{attribute addProperty BoxType "EK1122-0000-0018"}
{attribute addProperty Id "Beckhoff_EL30xxsub_EK1100EK1100_179A0949162"}
{attribute addProperty CRC "3537379036"}
{attribute addProperty SizeInBites "16"}
{attribute addProperty SizeInBytes "2"}
TYPE Beckhoff_EL30xxEK1122_D2D81EDC EXTENDS EK1122_179A0949 :
STRUCT
	{attribute addProperty Name "Beckhoff_EL30xxsub_EK1100"}
	Beckhoff_EL30xxsub_EK1100 : EK1100_179A0949;
END_STRUCT
END_TYPE

(* stored: Version 1.2.0.0, ProductVersion 3.1.4024.9
   DUT Beckhoff_EL30xxEK1122_D2D81EDC: Id {61a4f517-b592-48aa-9da4-e244fe614e53} *)
